PROGRAM MAIN
VAR
	i			: DINT;
END_VAR

i := i + 1;

END_PROGRAM

(* stored: Version 1.1.0.1, ProductVersion 3.1.4024.12
   POU MAIN: Id {98da3e34-4a61-4a8f-99e6-6cf9ea55f095}, SpecialFunc None *)
